(* IEC 61131-3 sources: 2026_Projet_YGO_ExcavatriceDragage/CODE_v0.5.25_20260807/SIMULATION, 2 files *)

(* ---- FB_Sim_Encoder.st ---- *)
(* ═══════════════════════════════════════════════════════════════
   🧪 FB_Sim_Encoder — Simulation physique d'un codeur absolu de treuil
   ───────────────────────────────────────────────────────────────
   📄 Doc métier : DOC/AF_Partie-13_Fonction_Simulation_v2.1.md
   🧩 Brique réduite (Partie3 §1bis, "briques E/S & diagnostics") : pas de contrat
      Enable/Reset/Error complet, pas de StartStop/SafeStop — outil de banc, pas
      du métier machine.
   🎯 Rôle : fait "compter" un codeur absolu comme si le treuil tournait
      réellement, à partir des relais de sens commandés et de la vitesse rampée
      courante. Extraction PURE de la logique déjà en place dans
      `PRG_02_Encoders.st` (bloc "SIMULATION SUR BANC DE TEST") — aucun
      changement de comportement, juste la dissociation en FB dédié.
   📥 Enable      : simulation active (SimulationModeActive AND NOT BusEncoderMxIsReal)
   📥 RelayFwd/RelayRev : sens commandé (contacteurs de sens du treuil)
   📥 SpeedRefPct : vitesse rampée courante (magnitude, %) — ex. instWinchM1.SpeedRamp.Current
   📥 PresetCmd   : TRUE le cycle où un preset (homing) doit être appliqué (PresettTrigCmd = 2)
   📥 PresetValue : valeur brute à charger lors du preset
   📥 SpeedScaleFactor : 🔧 REX 2026-07-07 — multiplicateur de vitesse simulation (confort de test
      banc uniquement, sans rapport avec une calibration réelle). Défaut 1.0 = comportement
      d'origine. Câblé sur GVL_Simulation.TstEncoderSpeedFactor (réglable à chaud, sans recompiler).
   📤 RawPosOut   : position brute simulée (UDINT), à aiguiller à la place de la valeur
      EtherCAT réelle quand le device n'est pas Operational (voir PRG_02_Encoders.st)
   🔧 REX 2026-07-08 : `RawPos` déplacé en `VAR_IN_OUT`, référencé depuis `GVL_PERSISTENT`
      (même pattern que `Calib` dans `FB_Encoder_Homing`) — `PERSISTENT` n'est valide que sur du
      `VAR_GLOBAL` en CODESYS, pas sur une variable locale de FB (tenté en `VAR RETAIN` puis
      `VAR PERSISTENT RETAIN` locaux, aucun des deux ne convient). Un vrai codeur absolu physique
      conserve son comptage brut même à travers un reset FROID (indépendant de l'automate) —
      il fallait donc bien du PERSISTENT RETAIN réel, regroupé avec le reste dans GVL_PERSISTENT.
   ═══════════════════════════════════════════════════════════════ *)

// === DECLARATION (à coller dans la partie déclaration du POU FB_Sim_Encoder) ===

FUNCTION_BLOCK PUBLIC FB_Sim_Encoder
VAR_INPUT
    Enable           : BOOL;
    RelayFwd         : BOOL;
    RelayRev         : BOOL;
    SpeedRefPct      : REAL;
    PresetCmd        : BOOL;
    PresetValue      : UDINT;
    SpeedScaleFactor : REAL := 1.0;   // 🔧 REX 2026-07-07 — confort de test, voir bandeau ci-dessus
    TestOffsetCmd    : BOOL;          // 🆕 REX 2026-07-08 (4) — front montant = applique TestOffsetPts (test banc)
    TestOffsetPts    : DINT := 0;     // 🆕 REX 2026-07-08 (4) — décalage signé à appliquer (points bruts)
END_VAR
VAR_OUTPUT
    RawPosOut   : UDINT;
END_VAR
VAR_IN_OUT
    RawPos      : UDINT;   // 🔧 REX 2026-07-08 : référence _SimEncoderRawPosM1/M2 (survit au reset froid)
END_VAR
VAR
    Increment      : UDINT;              // 🔧 REX 2026-07-07 — évite de dupliquer le calcul 2x
    TestOffsetEdge : R_TRIG;             // 🆕 REX 2026-07-08 (4)
END_VAR

// === IMPLEMENTATION (à coller dans le corps ST du POU FB_Sim_Encoder) ===

IF NOT Enable THEN
    RawPosOut := RawPos;
    RETURN;
END_IF;

// 🆕 REX 2026-07-08 (4) — injection test banc : VRAI saut de position (comme un glissement réel),
// pour tester Concept 1 / Méca E ET le rattrapage joystick (voir GVL_Simulation bandeau).
TestOffsetEdge(CLK := TestOffsetCmd);
IF TestOffsetEdge.Q THEN
    RawPos := DINT_TO_UDINT(UDINT_TO_DINT(RawPos) + TestOffsetPts);
END_IF;

Increment := REAL_TO_UDINT(SpeedRefPct * 0.1 * SpeedScaleFactor);

IF PresetCmd THEN
    RawPos := PresetValue;
ELSIF RelayFwd THEN
    RawPos := RawPos + Increment;
ELSIF RelayRev THEN
    IF RawPos >= Increment THEN
        RawPos := RawPos - Increment;
    ELSE
        RawPos := 0;
    END_IF;
END_IF;

RawPosOut := RawPos;

(* ---- FB_Sim_Safety.st ---- *)
(* ═══════════════════════════════════════════════════════════════
   🧪 FB_Sim_Safety — Simulation de la chaîne d'AU et du contacteur de puissance
   ───────────────────────────────────────────────────────────────
   📥 Enable          : activation de la simulation (SimulationModeActive AND NOT SensorEmergencyStopChainIsReal)
   📥 PowerCutOff_A   : demande de coupure PLC canal A (maintenu à TRUE en marche normale)
   📥 PowerCutOff_B   : demande de coupure PLC canal B (maintenu à TRUE en marche normale)
   📥 EmergencyArming : impulsion de réarmement (EmergencyArming_RQ)

   📤 SimChainOk      : simulation de la boucle AU (boutons relâchés et coupures PLC inactives)
   📤 SimContactorOk  : simulation du contacteur engagé (PowerContactorEngaged)

   ⚙️ Logique physique :
      - La chaîne d'AU (SimChainOk) est saine si les deux relais PLC de coupure sont maintenus fermés (TRUE).
      - Le contacteur s'engage (SimContactorOk) lors d'une impulsion de réarmement (EmergencyArming)
        et s'auto-maintient tant que la chaîne reste saine (SimChainOk).
      - Toute coupure de la chaîne (SimChainOk = FALSE) fait retomber immédiatement le contacteur.
   ═══════════════════════════════════════════════════════════════
   📄 Docs : DOC/AF_Partie-13_Fonction_Simulation_v2.1.md
*)
FUNCTION_BLOCK FB_Sim_Safety
VAR_INPUT
    Enable          : BOOL; // Activation de la simulation
    PowerCutOff_A   : BOOL; // Commande coupure canal A (TRUE = OK/fermé)
    PowerCutOff_B   : BOOL; // Commande coupure canal B (TRUE = OK/fermé)
    EmergencyArming : BOOL; // Impulsion de réarmement (TRUE = pulse)
    BtnEmergencyStop : BOOL; // Force l'ouverture de la boucle (TRUE = bouton appuyé/défaut)
END_VAR
VAR_OUTPUT
    SimChainOk      : BOOL; // Boucle AU simulée saine
    SimContactorOk  : BOOL; // Contacteur simulé engagé
END_VAR
VAR
    ContactorLatch  : BOOL; // Mémorisation de l'auto-maintien du contacteur
END_VAR

// === IMPLEMENTATION ===
IF NOT Enable THEN
    SimChainOk     := FALSE;
    SimContactorOk := FALSE;
    ContactorLatch := FALSE;
    RETURN;
END_IF;

// 1. La chaîne AU est saine si le PLC maintient les deux relais de coupure de puissance
// AND if no emergency stop button is pressed (BtnEmergencyStop is FALSE)
SimChainOk := PowerCutOff_A AND PowerCutOff_B AND NOT BtnEmergencyStop;

// 2. Logique d'auto-maintien (latch) du contacteur avec priorité à la coupure
IF NOT SimChainOk THEN
    ContactorLatch := FALSE;
ELSIF EmergencyArming THEN
    ContactorLatch := TRUE;
END_IF;

// Recopie vers la sortie
SimContactorOk := ContactorLatch;
